(* Copyright 2017 Cimpress

Licensed under the Apache License, Version 2.0 (the "License");
you may not use this file except in compliance with the License.
You may obtain a copy of the License at

http://www.apache.org/licenses/LICENSE-2.0

Unless required by applicable law or agreed to in writing, software
distributed under the License is distributed on an "AS IS" BASIS,
WITHOUT WARRANTIES OR CONDITIONS OF ANY KIND, either express or implied.
See the License for the specific language governing permissions and
limitations under the License. *)

TYPE E_SaberPlcDHCState :
(
	/// 0
	Init,
	/// 1
	WaitForData,
	/// 2
	RecvData,
	/// 3
	DataReady,
	/// 4
	Acknowledge,
	/// 5
	Retry,
	/// 6
	Error,
	/// 7
	WaitChannelInit,
	MAX_E_PlcSaberDHCStat
);
END_TYPE

(* stored: Version 1.1.0.1, ProductVersion 3.1.4019.2
   DUT E_SaberPlcDHCState: Id {1e18612b-6b33-4051-bacd-4a1469e1fae1} *)
